{attribute addProperty BoxType "EM7004-0000-0017"}
{attribute addProperty Id "OutputAT %Q*Output_BBA5775D162"}
{attribute addProperty CRC "1778418259"}
{attribute addProperty SizeInBites "16"}
{attribute addProperty SizeInBytes "2"}
TYPE DO_Outputs_6A008253 :
STRUCT
	{attribute addProperty Name "Output"}
	Output AT %Q* : Output_BBA5775D;
END_STRUCT
END_TYPE

(* stored: Version 1.2.0.0, ProductVersion 3.1.4024.9
   DUT DO_Outputs_6A008253: Id {905028d0-b835-457c-8a60-75ec25e609d3} *)
